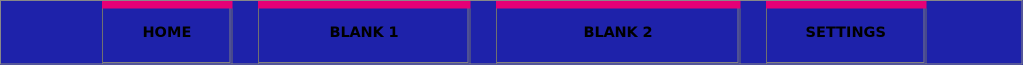
VISUALIZATION Navigation_Bar  // 1023x65
    Button (102,0 130x64), "HOME", image: JMTC.JMTC_Home_icon_32px
        tap HgV_Engine.stNav_Button[0].bToggle
    Button (258,0 212x64), "BLANK 1", image: JMTC.jmtc_sequence_icon_32px
        tap HgV_Engine.stNav_Button[1].bToggle
    Button (766,0 160x64), "SETTINGS", image: JMTC.jmtc_config_icon_32px
        tap HgV_Engine.stNav_Button[3].bToggle
    Rectangle (258,0 212x8), invisible if: HgV_Engine.stNav_Button[1].bInvisible
    Button (496,0 244x64), "BLANK 2", image: JMTC.jmtc_archive2_icon_32px
        tap HgV_Engine.stNav_Button[2].bToggle
    Rectangle (102,0 130x8), invisible if: HgV_Engine.stNav_Button[0].bInvisible
    Rectangle (496,0 244x8), invisible if: HgV_Engine.stNav_Button[2].bInvisible
    Rectangle (766,0 160x8), invisible if: HgV_Engine.stNav_Button[3].bInvisible
END_VISUALIZATION

(* stored: Version 1.1.0.1, ProductVersion 3.1.4022.18
   Visu Navigation_Bar: Id {b1495d13-4b96-46a3-9922-76e7162845a2} *)
